Universal Robots PolyScope program: Pick_Place_Exam.urp

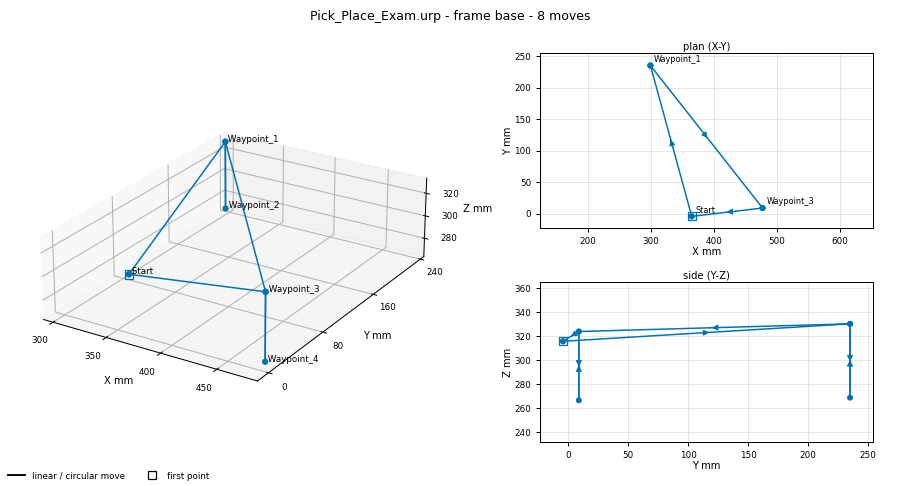
[picture p0: tool path of Pick_Place_Exam.urp in frame base, 8 of 8 moves have a stored position in this frame; points joined in program order, loops and branches not executed]
Program Pick_Place_Exam (installation=default directory=/programs/new folder createdIn=5.11.9.1010452 lastSavedIn=5.11.9.1010452 robotSerialNumber=20225200364)
Calibrated DH parameters: a=[0.00002, -0.569483, -0.54992, -0.00001, -0.000036, 0]; d=[0.180894, -146.691669, 192.918669, -46.053088, 0.119778, 0.115602]; alpha=[1.571425, -0.001534, 0.003359, 1.568739, -1.571477, 0]; deltaTheta=[0, 0.376258, -0.101074, -0.275185, -0.000002, 0]
Robot Program (runOnlyOnce=false)
  MoveL speed 250 mm/s, acceleration 1200 mm/s^2 (useActiveTCP=true) feature=Base
    Waypoint Start: TCP in base x=364.712 y=-4.206 z=315.757 mm, rx=-2.1744 ry=2.2654 rz=0.0306 rad; joints [27.5, -89.999, -129.437, 129.163, -91.268, -149.88] deg
    Waypoint Waypoint_1: TCP in base x=299.194 y=234.981 z=330.299 mm, rx=-2.1898 ry=2.242 rz=0.0149 rad; joints [65.296, -90.22, -127.131, -232.086, -90.525, -113.079] deg
    URCap RG Grip (OnRobot, OnRobot A/S) dataModel(rg-target-force=40.0, rg-target-width=0.1, Variable(key=on_return, variable(name=on_return)))
    Waypoint Waypoint_2: TCP in base x=299.219 y=234.98 z=268.769 mm, rx=-2.1896 ry=2.242 rz=0.0149 rad; joints [65.302, -95.072, -130.168, -224.191, -90.505, -113.044] deg
    URCap RG Grip (OnRobot, OnRobot A/S) dataModel(rg-target-force=40.0, rg-target-width=0.073)
    Waypoint Waypoint_1: TCP in base x=299.194 y=234.981 z=330.299 mm, rx=-2.1898 ry=2.242 rz=0.0149 rad; joints [65.296, -90.22, -127.131, -232.086, -90.525, -113.079] deg
    Waypoint Waypoint_3: TCP in base x=477.035 y=9.023 z=323.881 mm, rx=-2.1897 ry=2.242 rz=0.0149 rad; joints [22.322, -100.119, -116.94, -232.772, -90.829, -156.05] deg
    Waypoint Waypoint_4: TCP in base x=477.001 y=9.021 z=266.572 mm, rx=-2.1898 ry=2.2421 rz=0.0149 rad; joints [22.329, -104.04, -119.395, -226.403, -90.813, -156.023] deg
    URCap RG Grip (OnRobot, OnRobot A/S) dataModel(rg-target-force=40.0, rg-target-width=0.1)
    Waypoint Waypoint_3: TCP in base x=477.035 y=9.023 z=323.881 mm, rx=-2.1897 ry=2.242 rz=0.0149 rad; joints [22.322, -100.119, -116.94, -232.772, -90.829, -156.05] deg
    Waypoint Start: TCP in base x=364.712 y=-4.206 z=315.757 mm, rx=-2.1744 ry=2.2654 rz=0.0306 rad; joints [27.5, -89.999, -129.437, 129.163, -91.268, -149.88] deg
    Halt
